{attribute 'qualified_only'}
TYPE E_SystemType :
(
 	BekaPico,
	SkfETP2WZ
);
END_TYPE

(* stored: Version 1.1.0.1, ProductVersion 3.1.4024.12
   EnumerationTextList E_SystemType: Id {d2e6f4c0-f0c2-4f78-b107-bd808dbb0c0d} *)
